(* Logix 5000 project; controller water_tank vendor 1 type 14 code 150 rev 30.11; software revision 30.00 *)

TASK MainTask (continuous, watchdog 500 ms) : MainProgram

MODULES
   Local : vendor 1 type 14 code 150 (Compact 0, rev 30.11)
      Discrete_IO : Embedded (Compact 1, rev 3.1, Output RPI 20 ms)
      Analog_IO : Embedded (Compact 2, rev 1.1, Output RPI 80 ms)
      Counters : Embedded (Compact 3, rev 1.1, Output RPI 20 ms)
END_MODULES

PROGRAM MainProgram   (* main routine MainRoutine *)
VAR
   AUTO_READY : BOOL := 1;
   H_1 : ALIAS FOR Local:1:O.Data.7;   // HEATER TANK 2
   HEAT_R : REAL := 10485.0;
   HEAT_S : REAL := 80.11603;
   IR_1 : ALIAS FOR Local:1:I.Data.0;   // SENSOR 1
   IR_2 : ALIAS FOR Local:1:I.Data.1;   // SENSOR 2
   M_1 : ALIAS FOR Local:1:O.Data.5;   // PUMP MOTOR
   M_2 : ALIAS FOR Local:1:O.Data.6;   // CONVETOR MOTOR
   MAIN_R : REAL := 21000.0;
   MAIN_S : REAL := 25.862103;
   PB_1 : BOOL;   // FILL TANK ONE
   PB_2 : BOOL;   // FILL TANKN 2
   PB_3 : BOOL;   // DROP TANK ONE
   PB_4 : BOOL;   // DROP TANK TWO
   PB_5 : BOOL;   // CONVEYOR MOTOR
   PB_6 : BOOL;   // HEATER
   PL_1 : BOOL := 1;   // MANUAL LIGHT
   PL_2 : BOOL;   // AUTO LIGHT
   SOL_1 : ALIAS FOR Local:1:O.Data.0;   // FILL ONE
   SOL_2 : ALIAS FOR Local:1:O.Data.1;   // FILL TWO
   SOL_3 : ALIAS FOR Local:1:O.Data.2;   // DROP ONE
   SOL_4 : ALIAS FOR Local:1:O.Data.3;   // DROP TWO
   SW1 : BOOL;   // Auto/Manual
   TANK1_H : REAL := -2.0;
   TANK1_R : REAL := 18714.0;
   TANK1_S : REAL := 23.686043;
   TANK2_H : REAL := -2.0;
   TANK2_R : REAL := 14350.0;
   TANK2_S : REAL := 13.7320595;
   TANK_1_SP : REAL;   // Tank 1 Set-Point
   TANK_2_HT : REAL;   // Tank 2 Temp SP
   TANK_2_SP : REAL;   // Tank 2 Set-Point
   TEMP_H : REAL := -2.0;
END_VAR

ROUTINE auto   (* ladder *)
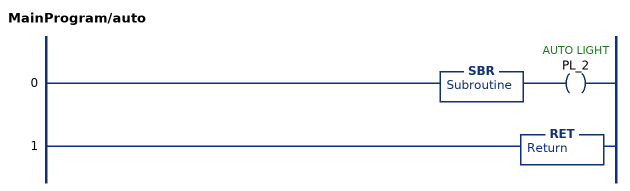
   0: SBR()OTE(PL_2);
   1: RET();
END_ROUTINE

ROUTINE MainRoutine   (* ladder *)
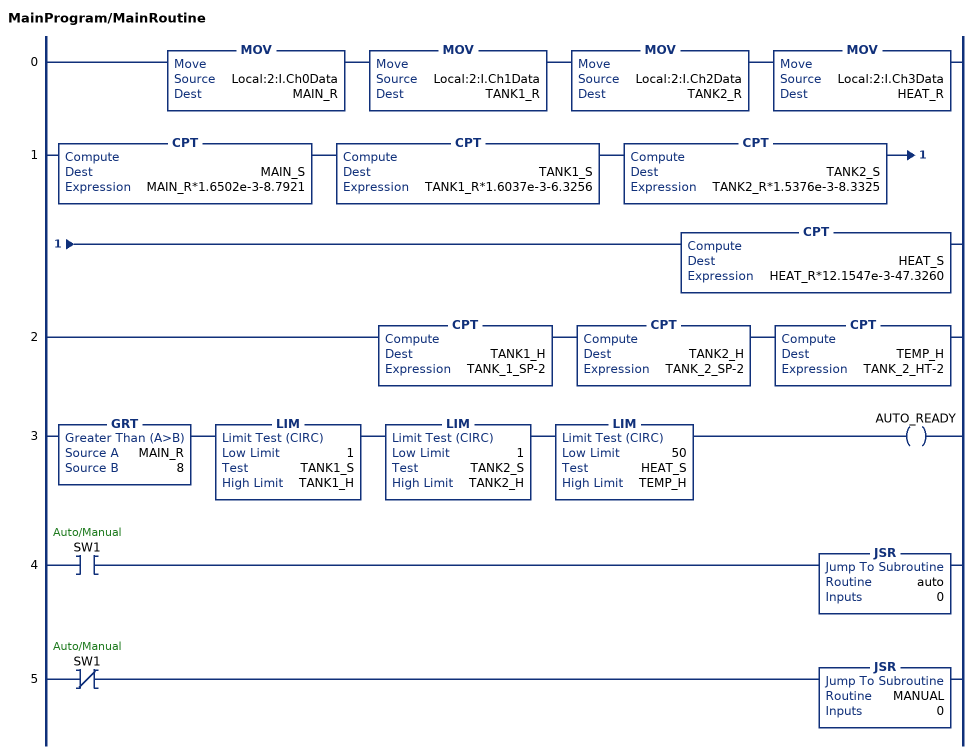
   0: MOV(Local:2:I.Ch0Data,MAIN_R)MOV(Local:2:I.Ch1Data,TANK1_R)MOV(Local:2:I.Ch2Data,TANK2_R)MOV(Local:2:I.Ch3Data,HEAT_R);
   1: CPT(MAIN_S,MAIN_R*1.6502e-3-8.7921)CPT(TANK1_S,TANK1_R*1.6037e-3-6.3256)CPT(TANK2_S,TANK2_R*1.5376e-3-8.3325)CPT(HEAT_S,HEAT_R*12.1547e-3-47.3260);
   2: CPT(TANK1_H,TANK_1_SP-2)CPT(TANK2_H,TANK_2_SP-2)CPT(TEMP_H,TANK_2_HT-2);
   3: GRT(MAIN_R,8)LIM(1,TANK1_S,TANK1_H)LIM(1,TANK2_S,TANK2_H)LIM(50,HEAT_S,TEMP_H)OTE(AUTO_READY);
   4: XIC(SW1)JSR(auto,0);
   5: XIO(SW1)JSR(MANUAL,0);
END_ROUTINE

ROUTINE MANUAL   (* ladder *)
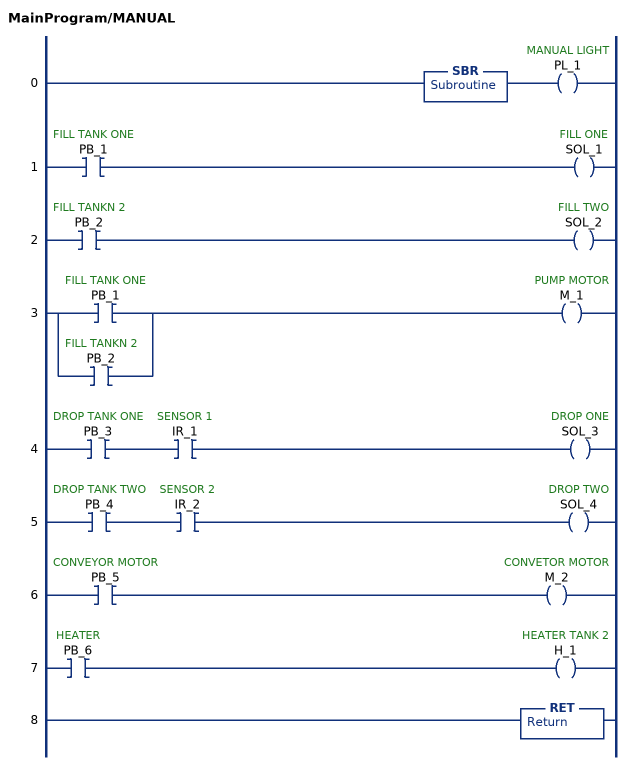
   0: SBR()OTE(PL_1);
   1: XIC(PB_1)OTE(SOL_1);
   2: XIC(PB_2)OTE(SOL_2);
   3: [XIC(PB_1) ,XIC(PB_2) ]OTE(M_1);
   4: XIC(PB_3)XIC(IR_1)OTE(SOL_3);
   5: XIC(PB_4)XIC(IR_2)OTE(SOL_4);
   6: XIC(PB_5)OTE(M_2);
   7: XIC(PB_6)OTE(H_1);
   8: RET();
END_ROUTINE
END_PROGRAM
